ACTION ACT_IO:
(*outputs*)
q_iRawPosition := iq_stVCN.q_iRawPosition;
(*inputs*)
iq_stVCN.i_iPosition := iq_stvcn.q_iRawPosition;
END_ACTION

END_FUNCTION_BLOCK

// POUs/Functions/Valves/FB_VFS
FUNCTION_BLOCK FB_VFS
(* This function block implements basic functionality for Fast Shutter/Valves*)
(* Fast Shutters do not function as complete isolation valves, but are intended to rapidly limit conductance 
between vacuum regions.  They should be installed in conjunction with isolation gate valves.  The conductance 
of the fast shutter in the closed state may be sufficiently low as to create an isolated vacuum region.  
Thus, at least a pirani gauge, that can measure a pressure down to 1x10-4 Torr, needs to be installed between
the shutter and the isolation gate valve.
In the case where a gauge is not installed, the neigboring gate Valves should not be opened unless the shutter 
is Open. 
*)
VAR_IN_OUT
	
END_VAR
VAR_INPUT
	{attribute 'pytmc' := 'pv: EPS_OK'}
	i_xEPS_OK:	BOOL	:= TRUE; (*External EPS interlock, Set to TRUE when no EPS interlock is required, otherwise set to correct interlock signal*)
	{attribute 'pytmc' := 'pv: PMPS_OK'}
	i_xPMPS_OK:	BOOL	; (*External MPS interlock, Set to TRUE when no PMPS interlock is required*)
	i_xExt_OK: BOOL; (*Other External Interlock, Set to True when no external interlock is required*)
	i_xOverrideMode : BOOL; (*To be linked to global override bit. This Overrides Vacuum logic only, EPS, MPS and PMPS are still enforces*)
END_VAR
VAR_OUTPUT
	{attribute 'pytmc' := '
    pv:
	'}
	iq_stValve : ST_VGC; (* All valve data and states will be in this struct*)
	
	{attribute 'pytmc' := 'pv: MPS_OK'}
	xMPS_OK:	BOOL; (*MPS Fast OK, is set when the Valve is Open*)
	
	
END_VAR
VAR
	rDiffPressAllowed	:	REAL := 22.5; // Torr, Default value comes from Vat Valve Manual
	rDiffPress : REAL;
	set : BOOL;
    reset: BOOL;
	  
	xFirstPass	:	BOOL;
	fbFSInit		:	R_TRIG;
	
	tonDelOK : TON;
	rtOK	:	R_TRIG;
	tonOvrd	:	TON;
	
	tDelOK	:	TIME := T#60S;
	tOvrd	:	TIME := T#10s;
	
	xClose: BOOL;
	CloseTimer: TON;
	TimDur: TIME := T#20MS;
	
	(* Timeouts*)
	tTimeOutDuration: TIME:= T#1S;
	tOPNtimeout: TON;
	tCLStimeout:TON;
	
	
	(*IO*)
	i_xOpnLS	AT%I*: BOOL;
	i_xClsLS	AT%I*: BOOL;
	q_xClose_A	AT%Q*: BOOL;
	q_xClose_B	AT%Q*: BOOL;
	q_xClose_C	AT%Q*: BOOL;
	q_xOPN_DO	AT%Q*: BOOL;
	i_xTrigger	AT%I*: BOOL; // Could be Up to 4
	{attribute 'pytmc' := 'pv: VAC_FAULT_OK'}
	xVAC_FAULT_OK AT%Q*: BOOL; (*Valve Vacuum OK, is set to Flase when there is Vacuum Fault*)
	
END_VAR

//TODO
// Make it better
//Test It
//Fix PVs and IO links
//Interface with neihboring valves.

(* Fast Shutter/Valve Function Block*)
(* M.Ghaly Feb 2019*)

(* Fast Shutters do not function as complete isolation valves, but are intended to rapidly limit conductance 
between vacuum regions.  They should be installed in conjunction with isolation gate valves.  The conductance 
of the fast shutter in the closed state may be sufficiently low as to create an isolated vacuum region.  
Thus, at least a pirani gauge, that can measure a pressure down to 1x10-4 Torr, needs to be installed between
the shutter and the isolation gate valve.
In the case where a gauge is not installed, the neigboring gate Valves should not be opened unless the shutter 
is Open. 
*)
(* Soft IO Mapping*)
IO();

///Check valve postion
IF iq_stValve.i_xClsLS AND  iq_stValve.i_xOpnLS THEN
	iq_stValve.eState:=INVALID;
ELSIF NOT iq_stValve.i_xClsLS AND iq_stValve.i_xOpnLS AND iq_stValve.q_xOPN_DO THEN 
	iq_stValve.eState:=OPEN;
ELSIF iq_stValve.i_xClsLS AND NOT iq_stValve.i_xOpnLS AND NOT iq_stValve.q_xOPN_DO THEN 
	iq_stValve.eState:=CLOSED;
ELSIF NOT iq_stValve.i_xClsLS AND NOT iq_stValve.i_xOpnLS THEN 
	iq_stValve.eState:=MOVING;
ELSE
	iq_stValve.eState:=INVALID;
END_IF

(* Input Trigger to close the Fast Shutter*)
(* Neighboring Valves Should also be triggered to Close*)
IF (i_xTrigger) THEN 
	xClose:= TRUE;
	xVAC_FAULT_OK:= FALSE;
	iq_stValve.xERR_LstVac := TRUE;
END_IF
IF (xClose) AND (NOT i_xClsLS) THEN
	q_xClose_A := TRUE;
	q_xClose_B := TRUE;
	q_xClose_C := TRUE;
END_IF
IF(CloseTimer.Q) OR (i_xClsLS) THEN
	q_xClose_A := FALSE;
	q_xClose_B := FALSE;
	q_xClose_C := FALSE;
	xClose := FALSE;
	iq_stValve.pv_xOPN_SW := FALSE;
END_IF

(* Neighboring Valves Interlock bit is reset When the Vacuum event error is reset and the Shutter is opened *)
IF (NOT i_xTrigger) AND (NOT iq_stValve.xERR_LstVac) AND i_xOpnLS THEN
	xVAC_FAULT_OK := TRUE;
END_IF

(*OPN OK evaluation bit *)
iq_stValve.xOPN_OK := (NOT iq_stValve.xERR_LstVac) AND NOT i_xTrigger;

(* If Epics Command to close the Valve, check if PMPS and EPS are ok, otherwise Keep command set to open valve *)
IF NOT(iq_stValve.pv_xOPN_SW) AND ((NOT i_xPMPS_OK) OR (NOT i_xEPS_OK) OR (NOT xVAC_FAULT_OK) ) THEN
	iq_stValve.pv_xOPN_SW := TRUE;
ELSE xClose := TRUE;
END_IF

(* Reset the EPICS command to open the valve if the interlock is lost *) 
(* based on EPS ok state, EPS overrides OPN_OK*)
IF NOT iq_stValve.xOPN_OK THEN
	IF i_xEPS_OK THEN iq_stValve.pv_xOPN_SW := FALSE;
	ELSE iq_stValve.pv_xOPN_SW := TRUE;		
	END_IF
END_IF

(* Here's where the valve opens *)
iq_stValve.q_xOPN_DO := (iq_stValve.pv_xOPN_SW AND iq_stValve.xOPN_OK) OR (tonOvrd.Q AND i_xOverrideMode);

(* When the valve  is open MPS is OK*)
xMPS_OK := (iq_stValve.eState=OPEN) AND NOT i_xTrigger;//??????


(* Override logic *)
(* Goal: give ability to override, but do so in a way that people won't forget it.
Solution: Override only after ten seconds of override, protect against blips,
when the valve permission goes true for more than ten seconds consistently, remove override
*)

tonDelOK(IN:=iq_stValve.xOPN_OK, PT:=tDelOK);
rtOK(CLK:=tonDelOK.Q);
IF rtOK.Q AND iq_stValve.pv_xOvrdOpn THEN 
	iq_stValve.pv_xOvrdOpn :=FALSE;
	iq_stValve.pv_xOPN_SW := TRUE; //for seamless transition
END_IF

//Override timer
tonOvrd(IN:=iq_stValve.pv_xOvrdOpn, PT:=tOvrd);



///Check valve postion timout
IF NOT iq_stValve.i_xClsLS AND tCLStimeout.Q THEN 
	iq_stValve.bErrorPresent := TRUE;
ELSIF NOT iq_stValve.i_xOpnLS AND tOPNtimeout.Q THEN 
	iq_stValve.bErrorPresent := TRUE;
END_IF

(*Timers*)
CloseTimer ( IN:=xClose, PT:= TimDur, Q=>);
tOPNtimeout(IN:= iq_stValve.q_xOPN_DO, PT := tTimeOutDuration );
tCLStimeout(IN:= NOT iq_stValve.q_xOPN_DO, PT := tTimeOutDuration);

(* Soft IO Mapping*)
IO();
// Alarm reset
//////////////////////////////////////
ACT_ResetAlarms();

ACTION ACT_ResetAlarms:
iq_stValve.xERR_DifPres R= iq_stValve.pv_xAlmRst;

iq_stValve.bErrorPresent R= iq_stValve.pv_xAlmRst;

IF NOT i_xTrigger THEN
	iq_stValve.xERR_LstVac R= iq_stValve.pv_xAlmRst;
END_IF
END_ACTION

ACTION IO:
(*inputs*)
iq_stValve.i_xOpnLS := 	i_xOpnLS;
iq_stValve.i_xClsLS:=	i_xClsLS;
iq_stValve.xEXT_OK := i_xEXT_OK;
iq_stValve.xOverrideMode := i_xOverrideMode;
(*outputs*)
q_xOPN_DO:= iq_stValve.q_xOPN_DO;
END_ACTION

END_FUNCTION_BLOCK

// POUs/Functions/Valves/FB_VGC
(* This function block implements basic functionality for Isolation Gate Valves*)
(* This function block interlock is as follows:
1. The valve can be opened when the difference between the pressures on both sides is
less than the maximum differential pressure.
2. This rule persists until the pressures on both sides are lower than the vacuum-setpoint.
3. Once at-vac, the valve will close if the pressure on either side rises above the setpoint.*)
(*This function block also implements PMPS and EPS interlocks, as well as Fast MPS trigger*)
FUNCTION_BLOCK FB_VGC
VAR_IN_OUT
	
END_VAR
VAR_INPUT
	(*Upstream Gauge, usually ion gauge*)
	i_stUSG	:	ST_VG;
	(*Downstream Gauge, usually ion gauge*)
	i_stDSG	:	ST_VG;
	{attribute 'pytmc' := '
    pv: Dis_DPIlk
	'}
	i_xDis_DPIlk : BOOL := FALSE;  (* Set to true when calling the function to disable the differential pressure interlock *)
	{attribute 'pytmc' := '
    pv: EPS_OK
	'}
	i_xEPS_OK:	BOOL	:= TRUE; (*External EPS interlock, Set to TRUE when no EPS interlock is required, otherwise set to correct interlock signal*)
	{attribute 'pytmc' := '
    pv: MPS_OK
	'}
	i_xPMPS_OK:	BOOL	; (*External MPS interlock, Set to TRUE when no PMPS interlock is required*)
	i_xExt_OK: BOOL; (*Other External Interlock, Set to True when no external interlock is required*)
	i_xOverrideMode : BOOL; (*To be linked to global override bit. This Overrides Vacuum logic only, EPS, MPS and PMPS are still enforces*)
END_VAR
VAR_OUTPUT
	{attribute 'pytmc' := '
    pv:
	'}
	iq_stValve : ST_VGC; (* All valve data and states will be in this struct*)
	
	{attribute 'pytmc' := '
    pv: MPS_FAULT
	'}
	xMPS_OK:	BOOL; (*MPS Fast OK, is set when the Valve is Open*)
END_VAR
VAR
	
	rDiffPressAllowed	:	REAL := 22.5; // Torr, Default value comes from Vat Valve Manual
	rDiffPress : REAL;
	set : BOOL;
    reset: BOOL;
	  
	xFirstPass	:	BOOL;
	fbFSInit		:	R_TRIG;
	
	tonDelOK : TON;
	rtOK	:	R_TRIG;
	tonOvrd	:	TON;
	
	tDelOK	:	TIME := T#60S;
	tOvrd	:	TIME := T#10s;
	
	
	(* Timeouts*)
	tTimeOutDuration: TIME:= T#5S;
	tOPNtimeout: TON;
	tCLStimeout:TON;
	
	
	(*IO*)
	i_xOpnLS	AT%I*: BOOL;
	i_xClsLS	AT%I*: BOOL;
	q_xOPN_DO	AT%Q*: BOOL;
	
END_VAR

(* Vacuum gate valve
A. Wallace
16-10-29

A gate valve isolates vacuum volumes. Ideally it can be opened when a system is vented
to allow for faster pumping, and will close when high vacuum is lost.

The following behavior is good for valves in something like a gas attenuator.
This function block does the following:
1. The valve can be opened when the difference between the pressures on both sides is
less than the maximum differential pressure.
2. This rule persists until the pressures on both sides are lower than the vacuum-setpoint.
3. Once at-vac, the valve will close if the pressure on either side rises above the setpoint.

Alternatively, the differential pressure interlock can be disabled so the valve may only be opened
if the pressure on both sides is lower than the at-vacuum-setpoint. You want this behavior if 
the valve is to be used in a UHV section.

Hysteresis is employed to ensure a smooth transition from vented/pumping down, to at-vac.

Finally, an override system is built in so you can bypass all the interlocking logic and 
get back online.
*)
(* 10/1/2018 Margaret Ghaly included EPS, PMPS Checkes and MPS trigger signals*)


fbFSInit( CLK := TRUE, Q => xFirstPass);
(*IO Mapping*)
ACT_IO();

(* On first PLC pass, put valve into vented state, which implies a closed valve *)
IF xFirstPass THEN
	iq_stValve.eVGC_State := Vented;
	iq_stValve.pv_xOPN_SW := FALSE;
END_IF


///Check valve postion
IF iq_stValve.i_xClsLS AND  iq_stValve.i_xOpnLS THEN
	iq_stValve.eState:=INVALID;
ELSIF NOT iq_stValve.i_xClsLS AND iq_stValve.i_xOpnLS AND iq_stValve.q_xOPN_DO THEN 
	iq_stValve.eState:=OPEN;
ELSIF iq_stValve.i_xClsLS AND NOT iq_stValve.i_xOpnLS AND NOT iq_stValve.q_xOPN_DO THEN 
	iq_stValve.eState:=CLOSED;
ELSIF NOT iq_stValve.i_xClsLS AND NOT iq_stValve.i_xOpnLS THEN 
	iq_stValve.eState:=MOVING;
ELSE
	iq_stValve.eState:=INVALID;
END_IF

// Update hysteresis
///////////////////////////////////////////////////
IF iq_stValve.rAT_VAC_SP_LAST <> iq_stValve.rAT_VAC_SP OR xFirstPass THEN
	iq_stValve.rAT_VAC_SP_LAST := iq_stValve.rAT_VAC_SP;
	iq_stValve.rAT_VAC_HYS := iq_stValve.rHYST_PERC * iq_stValve.rAT_VAC_SP;
END_IF

iq_stValve.rAT_VAC_HYS := LIMIT(0, iq_stValve.rAT_VAC_HYS, iq_stValve.rAT_VAC_SP);
IF iq_stValve.rAT_VAC_SP <> 0 THEN
	IF iq_stValve.rHYST_PERC <> (iq_stValve.rAT_VAC_HYS / iq_stValve.rAT_VAC_SP) THEN
		iq_stValve.rHYST_PERC := LIMIT(0, (iq_stValve.rAT_VAC_HYS / iq_stValve.rAT_VAC_SP) ,1);
	END_IF
END_IF
// Valve at vacuum check
///////////////////////////////////////////////////
	set := i_stUSG.rPRESS < iq_stValve.rAT_VAC_HYS AND i_stDSG.rPRESS < iq_stValve.rAT_VAC_HYS AND i_stUSG.xPRESS_OK AND i_stDSG.xPRESS_OK;
 	iq_stValve.xAT_VAC S= set;
	reset := i_stUSG.rPRESS > iq_stValve.rAT_VAC_SP OR i_stDSG.rPRESS > iq_stValve.rAT_VAC_SP OR NOT i_stUSG.xPRESS_OK OR NOT i_stDSG.xPRESS_OK;
	iq_stValve.xAT_VAC R= reset;
	
// Differential pressure check
///////////////////////////////////////////////////
	(* Calc the differential pressure across the valve *)
	rDiffPress := ABS(i_stUSG.rPRESS - i_stDSG.rPRESS);
	
	(* As long as the differential pressure is less than 30mbar, the valve is allowed to open *)
	IF rDiffPress <= rDiffPressAllowed AND i_stUSG.xPRESS_OK AND i_stDSG.xPRESS_OK THEN
		iq_stValve.xDP_OK := TRUE;
	ELSE
		iq_stValve.xDP_OK	:= FALSE;
		(* If the differential pressure is exceeded, even when the valve is open,
		the state is unexpected and triggers a fault, because it suggests that something
		is wrong with the valve, or gauges or mapping or there is a major leak on one side.*)
		iq_stValve.eVGC_State := ERR_DiffPress;
	END_IF

// Valve state
///////////////////////////////////////////////////
CASE iq_stValve.eVGC_State OF
	Vented: (* The Vented state is used during pump down *)
		(* Assuming the pump down went well, we are now at vacuum on both sides,
		so we move to the vacuum state, otherwise remain in the vented state *)
		IF iq_stValve.xAT_VAC THEN
		iq_stValve.eVGC_State := AtVacuum;
		ELSE
		iq_stValve.eVGC_State := Vented;
		END_IF
	
	AtVacuum:
		IF iq_stValve.xAT_VAC THEN
		(* If both pressure setpoints are made,
		then enable the differential pressure interlock, regardless of the valve state
		assuming we're using some kind of ion gauge where a pressure setpoint cannot be higher than 1E-4 T *)
		iq_stValve.eVGC_State := AtVacuum;
		ELSE
		
			(* If the valve is open (or in an unknown state) and either gauge is not at it's vacuum setpoint,
			we have a loss of vacuum error *)
			IF (iq_stValve.i_xOpnLS OR (NOT iq_stValve.i_xOpnLS AND NOT iq_stValve.i_xClsLS)) THEN
			iq_stValve.eVGC_State := ERR_LostVac;
		
			(* Alternatively, if the valve is already closed and we lose pressure on one side,
			it was probably intentional venting, so we calmly move back to venting mode, and
			disable the differential pressure interlock *) //?? 
			ELSIF iq_stValve.i_xClsLS THEN
			iq_stValve.eVGC_State := Vented;
			END_IF
		
		END_IF
	
	ERR_DiffPress:
		iq_stValve.eVGC_State := Vented;
		iq_stValve.xERR_DifPres := TRUE;
	
	ERR_LostVac:
		iq_stValve.eVGC_State := Vented;
		iq_stValve.xERR_LstVac := TRUE;
	
	END_CASE




// Interlock evaluation - with bypass for DP ILK bypass
///////////////////////////////////////////////
IF i_xDis_DPIlk THEN
	iq_stValve.xOPN_OK := iq_stValve.xEXT_OK; // AND iq_stValve.xDP_OK ;
ELSE
	iq_stValve.xOPN_OK := iq_stValve.xEXT_OK AND iq_stValve.xAT_VAC;
END_IF


(* Valve operation *)

(* Override logic *)
(* Goal: give ability to override, but do so in a way that people won't forget it.
Solution: Override only after ten seconds of override, protect against blips,
when the valve permission goes true for more than ten seconds consistently, remove override
*)

tonDelOK(IN:=iq_stValve.xOPN_OK, PT:=tDelOK);
rtOK(CLK:=tonDelOK.Q);
IF rtOK.Q AND iq_stValve.pv_xOvrdOpn THEN 
	iq_stValve.pv_xOvrdOpn :=FALSE;
	iq_stValve.pv_xOPN_SW := TRUE; //for seamless transition
END_IF

//Override timer
tonOvrd(IN:=iq_stValve.pv_xOvrdOpn, PT:=tOvrd);

(* If Epics Command to close the Valve, check if PMPS and EPS are ok, otherwise Keep command set to open valve *)
IF NOT(iq_stValve.pv_xOPN_SW) AND ((NOT i_xPMPS_OK) OR (NOT i_xEPS_OK)) THEN
	iq_stValve.pv_xOPN_SW := TRUE;
END_IF
(* Reset the EPICS command to open the valve if the interlock is lost *) 
(* based on EPS ok state, EPS overrides OPN_OK*)
IF NOT iq_stValve.xOPN_OK THEN
	IF i_xEPS_OK THEN iq_stValve.pv_xOPN_SW := FALSE;
	ELSE iq_stValve.pv_xOPN_SW := TRUE;		
	END_IF
END_IF

(* Here's where the valve opens *)
iq_stValve.q_xOPN_DO := (iq_stValve.pv_xOPN_SW AND iq_stValve.xOPN_OK) OR (tonOvrd.Q AND i_xOverrideMode);

(* When the valve  is open MPS is OK*)
xMPS_OK := (iq_stValve.eState=OPEN);//iq_stValve.i_xOpnLS; 

///Check valve moving postion timout
IF NOT iq_stValve.i_xClsLS AND tCLStimeout.Q THEN 
	iq_stValve.bErrorPresent := TRUE;
ELSIF NOT iq_stValve.i_xOpnLS AND tOPNtimeout.Q THEN 
	iq_stValve.bErrorPresent := TRUE; 
END_IF
IF (iq_stValve.eState=INVALID) THEN
	iq_stValve.bErrorPresent := TRUE; 
END_IF
(*Timers*)
tOPNtimeout(IN:= iq_stValve.q_xOPN_DO, PT := tTimeOutDuration );
tCLStimeout(IN:= NOT iq_stValve.q_xOPN_DO, PT := tTimeOutDuration);


// Alarm reset
//////////////////////////////////////
ACT_ResetAlarms();

(*IO Mapping*)
ACT_IO();

ACTION ACT_IO:
(*inputs*)
iq_stValve.i_xOpnLS := 	i_xOpnLS;
iq_stValve.i_xClsLS:=	i_xClsLS;
iq_stValve.xEXT_OK := i_xEXT_OK;
iq_stValve.xOverrideMode := i_xOverrideMode;
(*outputs*)
q_xOPN_DO:= iq_stValve.q_xOPN_DO;
END_ACTION

ACTION ACT_ResetAlarms:
iq_stValve.xERR_DifPres R= iq_stValve.pv_xAlmRst;
iq_stValve.xERR_LstVac R= iq_stValve.pv_xAlmRst;
iq_stValve.bErrorPresent R= iq_stValve.pv_xAlmRst;
END_ACTION

END_FUNCTION_BLOCK

// POUs/Functions/Valves/FB_VRC
(* This Function Block Implements Basic Functionality for certain types of valves e.g Turbo Isolation valves, Apperture Valve *)
(* Note Interlock Logic is External *)
FUNCTION_BLOCK FB_VRC
VAR_IN_OUT
	
END_VAR
VAR_INPUT
	i_xExtILK_OK : BOOL; //Connect to Interlock logic condition(e.g F_TURBO_VRC_ILK Function), otherwise, Set to True if the valve is not interlocked
	i_xOverrideMode : BOOL; (*To be linked to global override bit. This Overrides Vacuum logic only, EPS, MPS and PMPS are still enforces*)
END_VAR
VAR_OUTPUT
	{attribute 'pytmc' := '
    pv:
	'}
	iq_stValve : ST_VRC;
END_VAR
VAR

	tonOvrd	:	TON;
	tonDelOK : TON;
	rtOK	:	R_TRIG;

	(*IO*)
	i_xOpnLS	AT%I*: BOOL;
	i_xClsLS	AT%I*: BOOL;
	q_xOPN_DO	AT%Q*: BOOL;
END_VAR



///Check valve postion
IF NOT iq_stValve.i_xClsLS AND iq_stValve.i_xOpnLS THEN 
	iq_stValve.eState:=OPEN;
ELSIF iq_stValve.i_xClsLS AND NOT iq_stValve.i_xOpnLS THEN 
	iq_stValve.eState:=CLOSED;
ELSIF NOT iq_stValve.i_xClsLS AND NOT iq_stValve.i_xOpnLS THEN 
	iq_stValve.eState:=MOVING;
ELSE
	iq_stValve.eState:=INVALID;
END_IF

(*evaluate Valve open external interlock*)
iq_stValve.xOPN_OK := i_xExtILK_OK;
IF NOT iq_stValve.xOPN_OK and NOT tonOvrd.Q THEN
	iq_stValve.pv_xOPN_SW := FALSE;
END_IF

(* Override logic *)
(* Goal: give ability to override, but do so in a way that people won't forget it.
Solution: Override only after ten seconds of override, protect against blips,
when the valve permission goes true for more than ten seconds consistently, remove override
*)

tonDelOK(IN:=iq_stValve.xOPN_OK, PT:=T#10S);
rtOK(CLK:=tonDelOK.Q);
IF rtOK.Q THEN iq_stValve.pv_xOvrdOpn :=FALSE; END_IF

//Override timer
tonOvrd(IN:=iq_stValve.pv_xOvrdOpn, PT:=T#10S);

(* Here's where the valve opens *)
iq_stValve.q_xOPN_DO := (iq_stValve.pv_xOPN_SW AND iq_stValve.xOPN_OK) OR (tonOvrd.Q AND i_xOverrideMode);

(*Soft IO Mapping*)
ACT_IO();

ACTION ACT_IO:
(*inputs*)
iq_stValve.i_xOpnLS := 	i_xOpnLS;
iq_stValve.i_xClsLS:=	i_xClsLS;
iq_stValve.xOverrideMode := i_xOverrideMode;
(*outputs*)
q_xOPN_DO:= iq_stValve.q_xOPN_DO;
END_ACTION

END_FUNCTION_BLOCK

// POUs/Functions/Valves/FB_VRC_OK_CLS
(* This function block is different from the regular VRC in that CLOSING must be permitted. *)
FUNCTION_BLOCK FB_VRC_OK_CLS
VAR_IN_OUT
	iq_stValve : ST_VRC;
END_VAR
VAR_INPUT
	i_xOverrideMode : BOOL;
END_VAR
VAR_OUTPUT
END_VAR
VAR

tonOvrd	:	TON;
tonDelOK : TON;
rtOK	:	R_TRIG;

END_VAR

(* This function block is different from the regular VRC in that CLOSING must be permitted. *)
(* Implemented for the funky valve 04 on LAMP *)
IF NOT iq_stValve.xOPN_OK and NOT tonOvrd.Q THEN
iq_stValve.pv_xOPN_SW := FALSE;
END_IF

(* Override logic *)
(* Goal: give ability to override, but do so in a way that people won't forget it.
Solution: Override only after ten seconds of override, protect against blips,
when the valve permission goes true for more than ten seconds consistently, remove override
*)

tonDelOK(IN:=iq_stValve.xOPN_OK, PT:=T#10S);
rtOK(CLK:=tonDelOK.Q);
IF rtOK.Q THEN iq_stValve.pv_xOvrdOpn :=FALSE; END_IF

//Override timer
tonOvrd(IN:=iq_stValve.pv_xOvrdOpn, PT:=T#10S);

(* Here's where the valve opens *)
iq_stValve.q_xOPN_DO := NOT iq_stValve.xCLS_OK OR ((iq_stValve.pv_xOPN_SW AND iq_stValve.xOPN_OK) OR (tonOvrd.Q AND i_xOverrideMode));

END_FUNCTION_BLOCK

// POUs/Functions/Valves/FB_VVC
(* This Function Block Implements Basic Functionality for Vent Valves VVC *)
(* Note Interlock Logic is External *)
FUNCTION_BLOCK FB_VVC
VAR_IN_OUT

END_VAR
VAR_INPUT
	i_xExtILK_OK:BOOL; (*Other External Interlock, Set to True when no external interlock is required*)
	i_xOverrideMode : BOOL; (*To be linked to global override bit. This Overrides Vacuum logic only*)
END_VAR
VAR_OUTPUT
	{attribute 'pytmc' := '
    pv:
	'}
	iq_stValve : ST_VVC;
END_VAR
VAR

	tonOvrd	:	TON;
	tonDelOK : TON;
	rtOK	:	R_TRIG;

	(*IO*)
	q_xOPN_DO	AT%Q*: BOOL;

END_VAR


iq_stValve.xOPN_OK := i_xExtILK_OK;

IF NOT iq_stValve.xOPN_OK THEN
iq_stValve.pv_xOPN_SW := FALSE;
END_IF

(* Override logic *)
(* Goal: give ability to override, but do so in a way that people won't forget it.
Solution: Override only after ten seconds of override, protect against blips,
when the valve permission goes true for more than ten seconds consistently, remove override
*)

tonDelOK(IN:=iq_stValve.xOPN_OK, PT:=T#10S);
rtOK(CLK:=tonDelOK.Q);
IF rtOK.Q THEN iq_stValve.xOvrdOpn :=FALSE; END_IF

//Override timer
tonOvrd(IN:=iq_stValve.xOvrdOpn, PT:=T#10S);

(* Here's where the valve opens *)
iq_stValve.q_xOPN_DO := (iq_stValve.pv_xOPN_SW AND iq_stValve.xOPN_OK) OR (tonOvrd.Q AND i_xOverrideMode);

(*IO Mapping*)
ACT_IO();

ACTION ACT_IO:
(*inputs*)
iq_stValve.xOverrideMode := i_xOverrideMode;
(*outputs*)
q_xOPN_DO:= iq_stValve.q_xOPN_DO;
END_ACTION

END_FUNCTION_BLOCK
